RoboDK station: ObjectDeleter.rdk

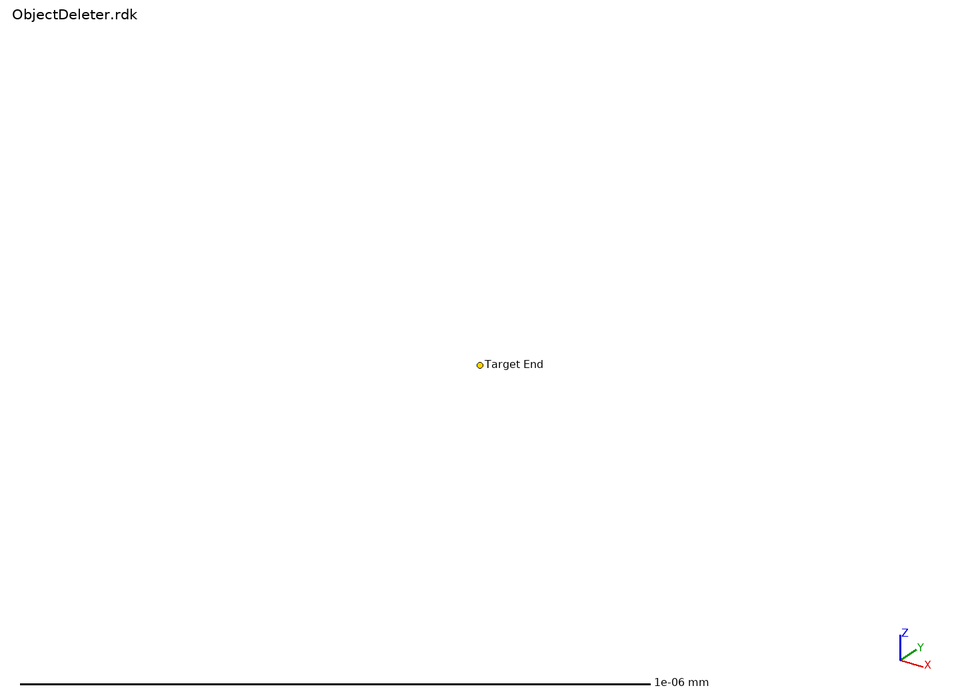
[picture v0: the station drawn from its stored meshes, robots at their saved joint values, targets as dots, program paths as lines]
Station ObjectDeleter (saved by RoboDK 5.5.4). Poses are relative to the parent item; angles as X-Y-Z fixed-axis rotations.
Station parameters (name, value as stored): Box-Spawner-Settings-0, Object-Deleter-Settings-0, Box-Spawner-Settings-0-Backup, Object-Deleter-Settings-0-Backup
  - frame Conveyor Belt Base at (500, 500, 0) mm
    - robot Conveyor Belt: 1 axes
        modified DH rows (alpha deg, a mm, theta deg, d mm): 0, 0, 0, 0 linear
        base shift (0, 0, 0) mm, rotated rx 0 ry 90 rz 0 deg
        joint limits [-500000] to [500000]; home [0]; saved at [-500000]
      - frame Conveyor Frame at (0, 0, 0) mm
    - frame Spawn Location at (0, 110, 0) mm
    - frame Delete Location at (1830, 110, 0) mm
    - target Target End (joint target) at (500000, 0, 0) mm; joints [500000] of Conveyor Belt
  - folder Scripts
    - Python program ConveyorReset (listed below)
    - Python program SpawnBox (listed below)
    - Python program DeleteObjects (listed below)
  - program SpawnerLoop (2 instructions, listed below)
  - program DeleterLoop (2 instructions, listed below)
  - program RunConveyor (2 instructions, listed below)
  - program Main (4 instructions, listed below)

--- Python program ConveyorReset ---
# Type help("robodk.robolink") or help("robodk.robomath") for more information
# Press F5 to run the script
# Documentation: https://robodk.com/doc/en/RoboDK-API.html
# Reference:     https://robodk.com/doc/en/PythonAPI/robodk.html
# Note: It is not required to keep a copy of this file, your Python script is saved with your RDK project

from robodk import robolink  # RoboDK API
from robodk import robomath  # Robot toolbox

#---------------------------------------
# Avoid auto-select
RDK = robolink.Robolink()
RDK.setSelection([])

#---------------------------------------
# Get the conveyor
conveyor = RDK.ItemUserPick(itemtype_or_list=robolink.ITEM_TYPE_ROBOT_AXES)
if not conveyor.Valid():
    quit()
conveyor_min, conveyor_max, _ = conveyor.JointLimits()

#---------------------------------------
# Get the conveyor's reference frame
frames = [x for x in conveyor.Childs() if x.Type() == robolink.ITEM_TYPE_FRAME]
conveyor_frame = frames[0]
if not conveyor_frame.Valid():
    quit()

#---------------------------------------
# Reset the conveyor
RDK.Render(False)
for child in conveyor_frame.Childs():
    if child.Type() == robolink.ITEM_TYPE_OBJECT and 'box' in child.Name().lower():
        child.Delete()
conveyor.setJoints(conveyor_min)
RDK.Render(True)

--- Python program SpawnBox ---
# --------------------------------------------
# --------------- DESCRIPTION ----------------
#
# Spawns a box using the preset settings.
# It can be called as an App action or within an App module.
#
# You can call it programmatically from a RoboDK program call.
# To use the spawner ID #2, call SpawnBox(2).
#
# More information about the RoboDK API for Python here:
#     https://robodk.com/doc/en/RoboDK-API.html
#     https://robodk.com/doc/en/PythonAPI/index.html
#
# More information on RoboDK Apps here:
#     https://github.com/RoboDK/Plug-In-Interface/tree/master/PluginAppLoader
#
# --------------------------------------------

from robodk import robolink, robomath, roboapps
import random
import os

try:
    from BoxSpawner import Settings  # Import as an App module. This is needed when the action is used externally, in a RoboDK script for instance.
except:
    import Settings


def SpawnBox(RDK=None, S=None):
    """
    Spawns a box using the preset settings.
    It can be called as an App action or within an App module.

    You can call it programmatically from a RoboDK program call.
    To use the spawner ID #2, call SpawnBox(2).
    """
    if RDK is None:
        RDK = robolink.Robolink()

    if S is None:
        S = Settings.Settings()
        S.Load(RDK)

    # Check if the parent exists
    PARENT_NAME = S.SPAWN_FRAME[1][S.SPAWN_FRAME[0]]
    PARENT = RDK.Item(PARENT_NAME)
    if not PARENT.Valid() or PARENT.Name() != PARENT_NAME or PARENT.Type() not in [robolink.ITEM_TYPE_STATION, robolink.ITEM_TYPE_FRAME]:
        RDK.ShowMessage(f"Unable to find the parent frame ({PARENT_NAME})! Did you set the settings?")
        return None

    # Check that the required files exists
    USE_METRIC = S.UNITS_TYPE[0] == 0

    # Attempt to recover the file location when used as a module
    if not os.path.exists(S.REF_BOX_MM_PATH):
        S.REF_BOX_MM_PATH = os.path.normpath(os.path.dirname(os.path.abspath(Settings.__file__)) + '/' + os.path.basename(S.REF_BOX_MM_PATH))
    if not os.path.exists(S.REF_BOX_IN_PATH):
        S.REF_BOX_IN_PATH = os.path.normpath(os.path.dirname(os.path.abspath(Settings.__file__)) + '/' + os.path.basename(S.REF_BOX_IN_PATH))

    if not USE_METRIC and not os.path.exists(S.REF_BOX_IN_PATH):
        RDK.ShowMessage(f"Unable to find the resource file ({S.REF_BOX_IN_PATH})!")
        return None
    elif USE_METRIC and not os.path.exists(S.REF_BOX_MM_PATH):
        RDK.ShowMessage(f"Unable to find the resource file ({S.REF_BOX_MM_PATH})!")
        return None

    RDK.Render(False)

    # Add the object
    if USE_METRIC:
        new_box = RDK.AddFile(S.REF_BOX_MM_PATH, PARENT)
    else:
        new_box = RDK.AddFile(S.REF_BOX_IN_PATH, PARENT)
    new_box.setVisible(False)

    # Set the initial size
    new_box.Scale(S.BOX_SIZE_XYZ)
    RDK.Update()

    # Randomize
    new_box.setPose(robomath.eye(4))
    pose = new_box.Pose()

    scale = 1.0
    if S.ENABLE_RANDOM_SIZE:
        scale = random.uniform(S.RANDOM_SIZE[0], S.RANDOM_SIZE[1])
        new_box.Scale(scale)
        RDK.Update()

    if S.ENABLE_RANDOM_POSITION:
        x = random.uniform(-S.RANDOM_POSITION[0], S.RANDOM_POSITION[0]) if S.RANDOM_POSITION[0] != 0. else 0.
        y = random.uniform(-S.RANDOM_POSITION[1], S.RANDOM_POSITION[1]) if S.RANDOM_POSITION[1] != 0. else 0.
        z = random.uniform(-S.RANDOM_POSITION[2], S.RANDOM_POSITION[2]) if S.RANDOM_POSITION[2] != 0. else 0.
        pose = robomath.RelTool(pose, x, y, z)

    if S.ENABLE_RANDOM_ORIENTATION:
        rx = random.uniform(-S.RANDOM_ORIENTATION[0], S.RANDOM_ORIENTATION[0]) if S.RANDOM_ORIENTATION[0] != 0. else 0.
        ry = random.uniform(-S.RANDOM_ORIENTATION[1], S.RANDOM_ORIENTATION[1]) if S.RANDOM_ORIENTATION[1] != 0. else 0.
        rz = random.uniform(-S.RANDOM_ORIENTATION[2], S.RANDOM_ORIENTATION[2]) if S.RANDOM_ORIENTATION[2] != 0. else 0.
        pose = robomath.RelTool(pose, 0, 0, 0, rx, ry, rz)

    new_box.setPose(pose)
    RDK.Update()

    # Set name according to new size
    sx, sy, sz = robomath.mult3(S.BOX_SIZE_XYZ, scale)
    new_box.setName((S.BOX_ITEM_NAME_MM if USE_METRIC else S.BOX_ITEM_NAME_IN) % (sx, sy, sz))

    # Attach to the closest conveyor
    if S.RELOCATE_TYPE[0] != 0:

        if S.RELOCATE_TYPE[0] == 1:
            # Closest conveyor
            parent_pos = PARENT.PoseAbs().Pos()
            conveyors = [x for x in RDK.ItemList(robolink.ITEM_TYPE_ROBOT_AXES) if len(x.Joints().tolist()) == 1]
            conveyors = sorted(conveyors, key=lambda x: robomath.distance(parent_pos, x.PoseAbs().Pos()))
            if not conveyors:
                RDK.ShowMessage("Unable to find any conveyor to attach too!")
                new_box.Delete()
                return None

            conveyor = conveyors[0]
            if robomath.distance(parent_pos, conveyor.PoseAbs().Pos()) > S.MAX_CONV_DISTANCE:
                RDK.ShowMessage("Unable to find any conveyor close enough to attach too ({S.MAX_CONV_DISTANCE} mm)!")
                new_box.Delete()
                return None

            frames = [x for x in conveyor.Childs() if x.Type() == robolink.ITEM_TYPE_FRAME]
            if not frames:
                frames = [RDK.AddFrame(conveyor.Name() + ' Frame', conveyor)]
            new_box.setParentStatic(frames[0])

        elif S.RELOCATE_TYPE[0] == 2:
            # Specific frame
            NEW_PARENT_NAME = S.RELOCATE_FRAME[1][S.RELOCATE_FRAME[0]]
            NEW_PARENT = RDK.Item(NEW_PARENT_NAME)
            if not NEW_PARENT.Valid() or NEW_PARENT.Name() != NEW_PARENT_NAME or NEW_PARENT.Type() not in [robolink.ITEM_TYPE_STATION, robolink.ITEM_TYPE_FRAME]:
                RDK.ShowMessage(f"Unable to find the parent frame ({NEW_PARENT_NAME})! Did you set the settings?")
                return None
            new_box.setParentStatic(NEW_PARENT)

    new_box.setVisible(True)
    RDK.Render(True)

    return new_box


def runmain():
    """
    Entrypoint of this action when it is executed on its own or interacted with in RoboDK.
    Important: Use the function name 'runmain()' if you want to compile this action.
    """

    if roboapps.Unchecked():
        roboapps.Exit()
    else:
        # When calling this script from a RoboDK Program, add the ID in the program call: SpawnBox(2)
        import sys
        id = 0
        if len(sys.argv) > 1:
            try:
                id = int(sys.argv[1])
            except:
                pass

        RDK = robolink.Robolink()

        S = Settings.Settings('Box-Spawner-Settings-' + str(id))
        S.Load(RDK)

        SpawnBox(RDK=RDK, S=S)


if __name__ == '__main__':
    runmain()

--- Python program DeleteObjects ---
# --------------------------------------------
# --------------- DESCRIPTION ----------------
#
# This file deletes objects in a zone using the preset settings.
# It can be called as an App action or within an App module.
#
# You can call it programmatically from a RoboDK program call.
# To use the zone ID #2, call DeleteObjectsLoop(2).
#
# More information about the RoboDK API for Python here:
#     https://robodk.com/doc/en/RoboDK-API.html
#     https://robodk.com/doc/en/PythonAPI/index.html
#
# More information on RoboDK Apps here:
#     https://github.com/RoboDK/Plug-In-Interface/tree/master/PluginAppLoader
#
# --------------------------------------------

from robodk import robolink, robomath, roboapps

try:
    from ObjectDeleter import Settings  # Import as an App module. This is needed when the action is used externally, in a RoboDK script for instance.
except:
    import Settings


def DeleteObjects(RDK=None, S=None):
    """
    This file deletes objects in a zone using the preset settings.
    It can be called as an App action or within an App module.

    You can call it programmatically from a RoboDK program call.
    To use the zone ID #2, call DeleteObjectsLoop(2).
    """
    if RDK is None:
        RDK = robolink.Robolink()

    if S is None:
        S = Settings.Settings()
        S.Load(RDK)

    # Check if the parent exists
    PARENT_NAME = S.ZONE_FRAME[1][S.ZONE_FRAME[0]]
    PARENT = RDK.Item(PARENT_NAME)
    if not PARENT.Valid() or PARENT.Name() != PARENT_NAME or PARENT.Type() not in [robolink.ITEM_TYPE_STATION, robolink.ITEM_TYPE_FRAME]:
        RDK.ShowMessage(f"Unable to find the parent frame ({PARENT_NAME})! Did you set the settings?")
        return False

    # Compile the regex, if any
    rgx = None
    if S.INCLUDE_REGEX:
        import re
        rgx = re.compile(S.INCLUDE_REGEX)

    # Get candidate items
    candidates = []
    if S.INCLUDE_OBJECT:
        candidates.extend(RDK.ItemList(robolink.ITEM_TYPE_OBJECT))
    if S.INCLUDE_CURVE:
        candidates.extend(RDK.ItemList(robolink.ITEM_TYPE_CURVE))
    if S.INCLUDE_FRAME:
        candidates.extend(RDK.ItemList(robolink.ITEM_TYPE_FRAME))
    if S.INCLUDE_TARGET:
        candidates.extend(RDK.ItemList(robolink.ITEM_TYPE_TARGET))

    # Find the items in the zone
    p_abs = PARENT.PoseAbs().Pos()
    objects = []
    for obj in candidates:
        if obj == PARENT:
            continue

        if not S.INCLUDE_HIDDEN and not obj.Visible():
            continue

        if rgx and not rgx.fullmatch(obj.Name()):
            continue

        if robomath.distance(p_abs, obj.PoseAbs().Pos()) > S.ZONE_RADIUS:
            continue

        objects.append(obj)

    # Delete the objects
    if objects:
        RDK.Render(False)
        RDK.Delete(objects)
        RDK.Render(True)

    return True


def runmain():
    """
    Entrypoint of this action when it is executed on its own or interacted with in RoboDK.
    Important: Use the function name 'runmain()' if you want to compile this action.
    """

    if roboapps.Unchecked():
        roboapps.Exit()
    else:
        # When calling this script from a RoboDK Program, add the ID in the program call: DeleteObjectsLoop(2)
        import sys
        id = 0
        if len(sys.argv) > 1:
            id = int(sys.argv[1])

        S = Settings.Settings('Object-Deleter-Settings-' + str(id))
        S.Load()

        DeleteObjects(S=S)


if __name__ == '__main__':
    runmain()

--- program SpawnerLoop (robot Conveyor Belt) ---
  Call SpawnBox(0)
  Pause 4.0 s

--- program DeleterLoop (robot Conveyor Belt) ---
  Call DeleteObjects(0)
  Pause 100 ms

--- program RunConveyor (robot Conveyor Belt) ---
  Set speed (100.0 mm/s)
  MoveJ (Target End)

--- program Main (robot Conveyor Belt) ---
  Call ConveyorReset
  Run RunConveyor
  Call SpawnerLoop
  Call DeleterLoop
